{attribute 'OPC.UA.DA.StructuredType' := '1'}
TYPE ST_SystemState :
STRUCT
	sOperatingState : STRING; //operating state (standby, operational, working)
	nOperatingState : E_SystemOperatingState; //operating state (standby, operational, working)
	bError : BOOL; //true if there is an error in any system component
END_STRUCT
END_TYPE

(* stored: Version 1.1.0.1, ProductVersion 3.1.4024.9
   DUT ST_SystemState: Id {e9d0f5d3-d47e-485c-a637-88ed8eb03f8a} *)
